KUKA KRL program: ab_a_lta_st01_g08.src, ab_a_lta_st01_g08.dat

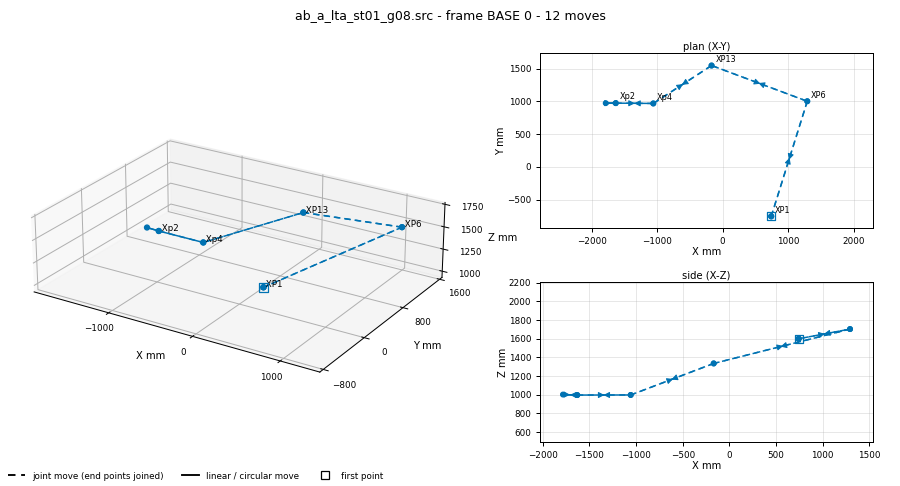
[picture p0: tool path of ab_a_lta_st01_g08.src in frame BASE 0, 12 of 12 moves have a stored position in this frame; points joined in program order, loops and branches not executed]
--- ab_a_lta_st01_g08.src ---
&ACCESS RVP1
&REL 10
&PARAM DISKPATH = KRC:\R1\Program\AXOR_ATEGO
DEF ab_a_lta_st01_g08( )

;FOLD INI;%{PE}
  ;FOLD BASISTECH INI
    GLOBAL INTERRUPT DECL 3 WHEN $STOPMESS==TRUE DO IR_STOPM ( )
    INTERRUPT ON 3
    BAS (#INITMOV,0 )
  ;ENDFOLD (BASISTECH INI)
;FOLD SPOTTECH INI
USERSPOT(#INIT)
;ENDFOLD (SPOTTECH INI)
;FOLD GRIPPERTECH INI
USER_GRP(0,DUMMY,DUMMY,GDEFAULT)
;ENDFOLD (GRIPPERTECH INI)
  ;FOLD USER INI
    ;Make your modifications here

  ;ENDFOLD (USER INI)
;ENDFOLD (INI)

;FOLD PTP P1 Vel=100 % PDAT1 Tool[5]:Gripper Geo G01 00 Base[0];%{PE}%R 8.2.24,%MKUKATPBASIS,%CMOVE,%VPTP,%P 1:PTP, 2:P1, 3:, 5:100, 7:PDAT1
$BWDSTART=FALSE
PDAT_ACT=PPDAT1
FDAT_ACT=FP1
BAS(#PTP_PARAMS,100)
PTP XP1
;ENDFOLD

; Caracterizacao dos meios de producao
; Changes: Deposita na Geo - ATEGO LTA
; Versao Atual: 28/12/2016
; Ferramenta: GRIPPER ATEGO/AXOR
; Name: P13.090-R6

chk_w5_wechs_ok ( )  ; CHECK GRP ATEGO

;FOLD PTP P5 Vel=100 % PDAT3 Tool[5]:Gripper Geo G01 00 Base[0];%{PE}%R 8.2.24,%MKUKATPBASIS,%CMOVE,%VPTP,%P 1:PTP, 2:P5, 3:, 5:100, 7:PDAT3
$BWDSTART=FALSE
PDAT_ACT=PPDAT3
FDAT_ACT=FP5
BAS(#PTP_PARAMS,100)
PTP XP5
;ENDFOLD

;FOLD ; Check Gripper GRAMPOS ABERTOS;%{PE}%R 8.2.24,%MKUKATPBASIS,%CCOMMENT,%VNORMAL,%P 2:Check Gripper GRAMPOS ABERTOS
;ENDFOLD
chk_w5_grp1_opn ()
chk_w5_grp2_opn ()
chk_w5_grp3_opn ()
chk_w5_grp4_opn ()

;FOLD ; Verifica GRIPPER SEM PECA;%{PE}%R 8.2.24,%MKUKATPBASIS,%CCOMMENT,%VNORMAL,%P 2:Verifica GRIPPER SEM PECA
;ENDFOLD
;FOLD WAIT FOR ( NOT IN 497 'Presenca peca 1 Axor/Atego' );%{PE}%R 8.2.24,%MKUKATPBASIS,%CEXT_WAIT_FOR,%VEXT_WAIT_FOR,%P 2:, 4:NOT, 5:$IN, 6:497, 7:Presenca peca 1 Axor/Atego, 9:
WAIT FOR  (  NOT $IN[497] )
;ENDFOLD
;FOLD WAIT FOR ( NOT IN 498 'Presenca peca 2 Axor/Atego' );%{PE}%R 8.2.24,%MKUKATPBASIS,%CEXT_WAIT_FOR,%VEXT_WAIT_FOR,%P 2:, 4:NOT, 5:$IN, 6:498, 7:Presenca peca 2 Axor/Atego, 9:
WAIT FOR  (  NOT $IN[498] )
;ENDFOLD

;FOLD ; Aguarda Liberacao p/ Encaixar no Painel Frontal ou Adiantamento;%{PE}%R 8.2.24,%MKUKATPBASIS,%CCOMMENT,%VNORMAL,%P 2:Aguarda Liberacao p/ Encaixar no  Painel Frontal ou Adiantamento
;ENDFOLD
;FOLD OUT 3347 'MAGAZINE 1 OCUPADO' State=TRUE ;%{PE}%R 8.2.24,%MKUKATPBASIS,%COUT,%VOUTX,%P 2:3347, 3:MAGAZINE 1 OCUPADO, 5:TRUE, 6:
$OUT[3347]=TRUE
;ENDFOLD
;FOLD OUT 3344 'APLICAÇÃO NÃO OK' State=TRUE ;%{PE}%R 8.2.24,%MKUKATPBASIS,%COUT,%VOUTX,%P 2:3344, 3:APLICAÇÃO NÃO OK, 5:TRUE, 6:
$OUT[3344]=TRUE
;ENDFOLD
;FOLD WAIT FOR ( IN 3347 'LIB. ANTECIPACAO (ATEGO/AXOR)' );%{PE}%R 8.2.24,%MKUKATPBASIS,%CEXT_WAIT_FOR,%VEXT_WAIT_FOR,%P 2:, 4:, 5:$IN, 6:3347, 7:LIB. ANTECIPACAO (ATEGO/AXOR), 9:
WAIT FOR  ( $IN[3347] )
;ENDFOLD
;FOLD OUT 3347 'MAGAZINE 1 OCUPADO' State=FALSE ;%{PE}%R 8.2.24,%MKUKATPBASIS,%COUT,%VOUTX,%P 2:3347, 3:MAGAZINE 1 OCUPADO, 5:FALSE, 6:
$OUT[3347]=FALSE
;ENDFOLD

;FOLD PTP P6 CONT Vel=100 % PDAT4 Tool[5]:Gripper Geo G01 00 Base[0];%{PE}%R 8.2.24,%MKUKATPBASIS,%CMOVE,%VPTP,%P 1:PTP, 2:P6, 3:C_PTP, 5:100, 7:PDAT4
$BWDSTART=FALSE
PDAT_ACT=PPDAT4
FDAT_ACT=FP6
BAS(#PTP_PARAMS,100)
PTP XP6 C_PTP
;ENDFOLD
;FOLD PTP P13 CONT Vel=100 % PDAT5 Tool[5]:Gripper Geo G01 00 Base[0];%{PE}%R 8.2.24,%MKUKATPBASIS,%CMOVE,%VPTP,%P 1:PTP, 2:P13, 3:C_PTP, 5:100, 7:PDAT5
$BWDSTART=FALSE
PDAT_ACT=PPDAT5
FDAT_ACT=FP13
BAS(#PTP_PARAMS,100)
PTP XP13 C_PTP
;ENDFOLD
;FOLD PTP p4 CONT Vel=100 % P_OLP3 Tool[5]:Gripper Geo G01 00 Base[0];%{PE}%R 8.2.24,%MKUKATPBASIS,%CMOVE,%VPTP,%P 1:PTP, 2:p4, 3:C_PTP, 5:100, 7:P_OLP3
$BWDSTART=FALSE
PDAT_ACT=PP_OLP3
FDAT_ACT=Fp4
BAS(#PTP_PARAMS,100)
PTP Xp4 C_PTP
;ENDFOLD

;FOLD ; Aguarda Liberacao p/ Encaixar GRIPPER no Painel Frontal;%{PE}%R 8.2.24,%MKUKATPBASIS,%CCOMMENT,%VNORMAL,%P 2:Aguarda Liberacao p/ Encaixar GRIPPER no Painel Frontal
;ENDFOLD
;FOLD WAIT FOR ( IN 3344 'LIB.P/APOIO DO TETO (ATEGO/AXOR)' );%{PE}%R 8.2.24,%MKUKATPBASIS,%CEXT_WAIT_FOR,%VEXT_WAIT_FOR,%P 2:, 4:, 5:$IN, 6:3344, 7:LIB.P/APOIO DO TETO (ATEGO/AXOR), 9:
WAIT FOR  ( $IN[3344] )
;ENDFOLD
;FOLD OUT 3344 'APLICAÇÃO NÃO OK' State=FALSE ;%{PE}%R 8.2.24,%MKUKATPBASIS,%COUT,%VOUTX,%P 2:3344, 3:APLICAÇÃO NÃO OK, 5:FALSE, 6:
$OUT[3344]=FALSE
;ENDFOLD

;FOLD LIN p2 Vel=0.25 m/s L_OLP1 Tool[5]:Gripper Geo G01 00 Base[0];%{PE}%R 8.2.24,%MKUKATPBASIS,%CMOVE,%VLIN,%P 1:LIN, 2:p2, 3:, 5:0.25, 7:L_OLP1
$BWDSTART=FALSE
LDAT_ACT=LL_OLP1
FDAT_ACT=Fp2
BAS(#CP_PARAMS,0.25)
LIN Xp2
;ENDFOLD

;FOLD ; Posicao Geometria Gripper ATEGO/AXOR;%{PE}%R 8.2.24,%MKUKATPBASIS,%CCOMMENT,%VNORMAL,%P 2:Posicao Geometria Gripper ATEGO/AXOR
;ENDFOLD
;FOLD LIN P14 Vel=0.15 m/s CPDAT1 Tool[5]:Gripper Geo G01 00 Base[0];%{PE}%R 8.2.24,%MKUKATPBASIS,%CMOVE,%VLIN,%P 1:LIN, 2:P14, 3:, 5:0.15, 7:CPDAT1
$BWDSTART=FALSE
LDAT_ACT=LCPDAT1
FDAT_ACT=FP14
BAS(#CP_PARAMS,0.15)
LIN XP14
;ENDFOLD

;FOLD ; Fechar Grampos Z4,Z2 e Z1;%{PE}%R 8.2.24,%MKUKATPBASIS,%CCOMMENT,%VNORMAL,%P 2:Fechar Grampos Z4,Z2 e Z1
;ENDFOLD
;FOLD SET GRP 4 State=CLO GDAT6;%{PE}%R 8.2.4,%MKUKATPGRP,%CGRP,%VGRP,%P 2:4, 4:1, 5:#NO, 6:GDAT6, 8:0, 10:0
H50(GRP,4,1,GGDAT6)
;ENDFOLD
chk_w5_grp4_clo ()
;FOLD SET GRP 1 State=CLO GDAT2;%{PE}%R 8.2.4,%MKUKATPGRP,%CGRP,%VGRP,%P 2:1, 4:1, 5:#NO, 6:GDAT2, 8:0, 10:0
H50(GRP,1,1,GGDAT2)
;ENDFOLD
;FOLD SET GRP 2 State=CLO GDAT3;%{PE}%R 8.2.4,%MKUKATPGRP,%CGRP,%VGRP,%P 2:2, 4:1, 5:#NO, 6:GDAT3, 8:0, 10:0
H50(GRP,2,1,GGDAT3)
;ENDFOLD
;FOLD ; Aguarda Grampos Z1 e Z2 FECHADOS e Z3 ABERTO;%{PE}%R 8.2.24,%MKUKATPBASIS,%CCOMMENT,%VNORMAL,%P 2:Aguarda Grampos Z1 e Z2 FECHADOS e Z3 ABERTO
;ENDFOLD
chk_w5_grp1_clo ()
chk_w5_grp2_clo ()
chk_w5_grp3_opn ()

;FOLD ; Verifica garra com peca;%{PE}%R 8.2.24,%MKUKATPBASIS,%CCOMMENT,%VNORMAL,%P 2:Verifica  garra  com  peca
;ENDFOLD
IF (NOT(GHOST())) THEN
;FOLD WAIT FOR ( IN 497 'Presenca peca 1 Axor/Atego' );%{PE}%R 8.2.24,%MKUKATPBASIS,%CEXT_WAIT_FOR,%VEXT_WAIT_FOR,%P 2:, 4:, 5:$IN, 6:497, 7:Presenca peca 1 Axor/Atego, 9:
WAIT FOR  ( $IN[497] )
;ENDFOLD
;FOLD WAIT FOR ( IN 498 'Presenca peca 2 Axor/Atego' );%{PE}%R 8.2.24,%MKUKATPBASIS,%CEXT_WAIT_FOR,%VEXT_WAIT_FOR,%P 2:, 4:, 5:$IN, 6:498, 7:Presenca peca 2 Axor/Atego, 9:
WAIT FOR  ( $IN[498] )
;ENDFOLD
ENDIF

;FOLD ; Robo na posicao;%{PE}%R 8.2.24,%MKUKATPBASIS,%CCOMMENT,%VNORMAL,%P 2:Robo  na  posicao
;ENDFOLD
;FOLD OUT 3345 'ALERTA DE APLICAÇÃO' State=TRUE ;%{PE}%R 8.2.24,%MKUKATPBASIS,%COUT,%VOUTX,%P 2:3345, 3:ALERTA DE APLICAÇÃO, 5:TRUE, 6:
$OUT[3345]=TRUE
;ENDFOLD

;FOLD ; Aguarda liberacao para sair com a garra;%{PE}%R 8.2.24,%MKUKATPBASIS,%CCOMMENT,%VNORMAL,%P 2:Aguarda  liberacao  para  sair  com  a  garra
;ENDFOLD
;FOLD WAIT FOR ( IN 3345 'LIB.SAÍDA APOIO DO TETO (ATEGO/AXOR)' );%{PE}%R 8.2.24,%MKUKATPBASIS,%CEXT_WAIT_FOR,%VEXT_WAIT_FOR,%P 2:, 4:, 5:$IN, 6:3345, 7:LIB.SAÍDA APOIO DO TETO (ATEGO/AXOR), 9:
WAIT FOR  ( $IN[3345] )
;ENDFOLD
;FOLD OUT 3345 'ALERTA DE APLICAÇÃO' State=FALSE ;%{PE}%R 8.2.24,%MKUKATPBASIS,%COUT,%VOUTX,%P 2:3345, 3:ALERTA DE APLICAÇÃO, 5:FALSE, 6:
$OUT[3345]=FALSE
;ENDFOLD

;FOLD ; Abrir grampos Z1,Z2,Z4;%{PE}%R 8.2.24,%MKUKATPBASIS,%CCOMMENT,%VNORMAL,%P 2:Abrir  grampos  Z1,Z2,Z4
;ENDFOLD
;FOLD SET GRP 1 State=OPN GDAT1;%{PE}%R 8.2.4,%MKUKATPGRP,%CGRP,%VGRP,%P 2:1, 4:2, 5:#NO, 6:GDAT1, 8:0, 10:0
H50(GRP,1,2,GGDAT1)
;ENDFOLD
;FOLD SET GRP 2 State=OPN GDAT7;%{PE}%R 8.2.4,%MKUKATPGRP,%CGRP,%VGRP,%P 2:2, 4:2, 5:#NO, 6:GDAT7, 8:0, 10:0
H50(GRP,2,2,GGDAT7)
;ENDFOLD
;FOLD SET GRP 3 State=OPN GDAT8;%{PE}%R 8.2.4,%MKUKATPGRP,%CGRP,%VGRP,%P 2:3, 4:2, 5:#NO, 6:GDAT8, 8:0, 10:0
H50(GRP,3,2,GGDAT8)
;ENDFOLD
;FOLD SET GRP 4 State=OPN GDAT9;%{PE}%R 8.2.4,%MKUKATPGRP,%CGRP,%VGRP,%P 2:4, 4:2, 5:#NO, 6:GDAT9, 8:0, 10:0
H50(GRP,4,2,GGDAT9)
;ENDFOLD
chk_w5_grp1_opn ()
chk_w5_grp2_opn ()
chk_w5_grp3_opn ()
chk_w5_grp4_opn ()

;FOLD LIN P15 Vel=0.15 m/s CPDAT2 Tool[5]:Gripper Geo G01 00 Base[0];%{PE}%R 8.2.24,%MKUKATPBASIS,%CMOVE,%VLIN,%P 1:LIN, 2:P15, 3:, 5:0.15, 7:CPDAT2
$BWDSTART=FALSE
LDAT_ACT=LCPDAT2
FDAT_ACT=FP15
BAS(#CP_PARAMS,0.15)
LIN XP15
;ENDFOLD

;FOLD WAIT FOR ( NOT IN 497 'Presenca peca 1 Axor/Atego' );%{PE}%R 8.2.24,%MKUKATPBASIS,%CEXT_WAIT_FOR,%VEXT_WAIT_FOR,%P 2:, 4:NOT, 5:$IN, 6:497, 7:Presenca peca 1 Axor/Atego, 9:
WAIT FOR  (  NOT $IN[497] )
;ENDFOLD
;FOLD WAIT FOR ( NOT IN 498 'Presenca peca 2 Axor/Atego' );%{PE}%R 8.2.24,%MKUKATPBASIS,%CEXT_WAIT_FOR,%VEXT_WAIT_FOR,%P 2:, 4:NOT, 5:$IN, 6:498, 7:Presenca peca 2 Axor/Atego, 9:
WAIT FOR  (  NOT $IN[498] )
;ENDFOLD

;FOLD PTP P0 Vel=100 % P_OLP7 Tool[5]:Gripper Geo G01 00 Base[0];%{PE}%R 8.2.24,%MKUKATPBASIS,%CMOVE,%VPTP,%P 1:PTP, 2:P0, 3:, 5:100, 7:P_OLP7
$BWDSTART=FALSE
PDAT_ACT=PP_OLP7
FDAT_ACT=FP0
BAS(#PTP_PARAMS,100)
PTP XP0
;ENDFOLD
;FOLD PTP p9 CONT Vel=100 % P_OLP5 Tool[5]:Gripper Geo G01 00 Base[0];%{PE}%R 8.2.24,%MKUKATPBASIS,%CMOVE,%VPTP,%P 1:PTP, 2:p9, 3:C_PTP, 5:100, 7:P_OLP5
$BWDSTART=FALSE
PDAT_ACT=PP_OLP5
FDAT_ACT=Fp9
BAS(#PTP_PARAMS,100)
PTP Xp9 C_PTP
;ENDFOLD
;FOLD PTP p12 CONT Vel=100 % P_OLP6 Tool[5]:Gripper Geo G01 00 Base[0];%{PE}%R 8.2.24,%MKUKATPBASIS,%CMOVE,%VPTP,%P 1:PTP, 2:p12, 3:C_PTP, 5:100, 7:P_OLP6
$BWDSTART=FALSE
PDAT_ACT=PP_OLP6
FDAT_ACT=Fp12
BAS(#PTP_PARAMS,100)
PTP Xp12 C_PTP
;ENDFOLD
;FOLD PTP P16 Vel=100 % PDAT6 Tool[5]:Gripper Geo G01 00 Base[0];%{PE}%R 8.2.24,%MKUKATPBASIS,%CMOVE,%VPTP,%P 1:PTP, 2:P16, 3:, 5:100, 7:PDAT6
$BWDSTART=FALSE
PDAT_ACT=PPDAT6
FDAT_ACT=FP16
BAS(#PTP_PARAMS,100)
PTP XP16
;ENDFOLD

;FOLD ; Libera dispositivo para soldar respot;%{PE}%R 8.2.24,%MKUKATPBASIS,%CCOMMENT,%VNORMAL,%P 2:Libera  dispositivo  para  soldar  respot
;ENDFOLD
;FOLD OUT 3347 'MAGAZINE 1 OCUPADO' State=TRUE ;%{PE}%R 8.2.24,%MKUKATPBASIS,%COUT,%VOUTX,%P 2:3347, 3:MAGAZINE 1 OCUPADO, 5:TRUE, 6:
$OUT[3347]=TRUE
;ENDFOLD
;FOLD OUT 3344 'APLICAÇÃO NÃO OK' State=TRUE ;%{PE}%R 8.2.24,%MKUKATPBASIS,%COUT,%VOUTX,%P 2:3344, 3:APLICAÇÃO NÃO OK, 5:TRUE, 6:
$OUT[3344]=TRUE
;ENDFOLD

;FOLD PULSE 3340 'R6 GEOMETRIA OK' State=TRUE Time=1 sec;%{PE}%R 8.2.24,%MKUKATPBASIS,%COUT,%VPULSE,%P 2:3340, 3:R6 GEOMETRIA OK, 5:TRUE, 6:, 8:1
PULSE($OUT[3340], TRUE,1)
;ENDFOLD
END

--- ab_a_lta_st01_g08.dat ---
&ACCESS RVP1
&REL 10
&PARAM DISKPATH = KRC:\R1\Program\AXOR_ATEGO
DEFDAT  ab_a_lta_st01_g08
;FOLD EXTERNAL DECLARATIONS;%{PE}%MKUKATPBASIS,%CEXT,%VCOMMON,%P
;FOLD BASISTECH EXT;%{PE}%MKUKATPBASIS,%CEXT,%VEXT,%P
EXT  BAS (BAS_COMMAND  :IN,REAL  :IN )
DECL INT SUCCESS
;ENDFOLD (BASISTECH EXT)
;FOLD USER EXT;%{E}%MKUKATPUSER,%CEXT,%VEXT,%P
;Make your modifications here
;ENDFOLD (USER EXT)
;ENDFOLD (EXTERNAL DECLARATIONS)

;# ============ START PATH : ab_a_lta_st01_g08 =============
DECL FDAT Fp11={TOOL_NO 5,BASE_NO 0,IPO_FRAME #BASE,POINT2[] " "}
DECL PDAT PP_OLP1={VEL 100.0,ACC 100.0,APO_DIST 0.0}
DECL E6POS Xp11={X 1293.05103,Y 1000.521,Z 1703.34399,A 36.1688995,B -6.9552002,C 153.792801,S 6,T 19}
DECL FDAT Fp10={TOOL_NO 5,BASE_NO 0,IPO_FRAME #BASE,POINT2[] " "}
DECL PDAT PP_OLP2={VEL 100.0,ACC 100.0,APO_DIST 0.0}
DECL E6POS Xp10={X -168.237,Y 1546.06995,Z 1335.04004,A 110.0187,B -0.406599998,C 159.128998,S 6,T 19}
DECL FDAT Fp4={TOOL_NO 5,BASE_NO 0,IPO_FRAME #BASE,POINT2[] " "}
DECL PDAT PP_OLP3={VEL 100.0,ACC 20.0,APO_DIST 0.0,APO_MODE #CPTP}
DECL E6POS Xp4={X -1057.83704,Y 966.953003,Z 997.169983,A -179.672195,B -1.48539996,C 179.896301,S 6,T 19}
DECL FDAT Fp2={TOOL_NO 5,BASE_NO 0,IPO_FRAME #BASE,POINT2[] " "}
DECL E6POS Xp2={X -1631.20996,Y 971.839417,Z 996.094482,A -179.828995,B -0.654202104,C 179.611496,S 22,T 19,E1 0.0,E2 0.0,E3 0.0,E4 0.0,E5 0.0,E6 0.0}
DECL LDAT LL_OLP1={VEL 0.25,ACC 100.0,APO_DIST 0.0,APO_FAC 0.0,ORI_TYP #VAR,CIRC_TYP #BASE,JERK_FAC 50.0}
DECL FDAT Fl005={TOOL_NO 5,BASE_NO 0,IPO_FRAME #BASE,POINT2[] " "}
DECL E6POS Xl005={X -1795.66003,Y 969.495972,Z 1016.79303,A 179.821594,B -1.35329998,C 179.764893,S 6,T 19}
DECL LDAT LL_OLP2={VEL 0.100000001,ACC 100.0,APO_DIST 0.0,APO_FAC 0.0,ORI_TYP #VAR,CIRC_TYP #BASE,JERK_FAC 50.0}
DECL FDAT Fp7={TOOL_NO 5,BASE_NO 0,IPO_FRAME #BASE,POINT2[] " "}
DECL E6POS Xp7={X -1650.26294,Y 963.580017,Z 1010.07397,A -179.672302,B -1.48520005,C 179.896301,S 6,T 19}
DECL LDAT LL_OLP3={VEL 0.25,ACC 100.0,APO_DIST 0.0,APO_FAC 0.0,ORI_TYP #VAR,CIRC_TYP #BASE,JERK_FAC 50.0}
DECL FDAT Fp8={TOOL_NO 5,BASE_NO 0,IPO_FRAME #BASE,POINT2[] " "}
DECL PDAT PP_OLP4={VEL 100.0,ACC 100.0,APO_DIST 0.0}
DECL E6POS Xp8={X -1057.83704,Y 966.953003,Z 997.169983,A -179.672302,B -1.48539996,C 179.896301,S 6,T 19}
DECL FDAT Fp9={TOOL_NO 5,BASE_NO 0,IPO_FRAME #BASE,POINT2[] " "}
DECL PDAT PP_OLP5={VEL 100.0,ACC 20.0,APO_DIST 20.0,APO_MODE #CPTP}
DECL E6POS Xp9={X -168.237,Y 1546.06995,Z 1335.04004,A 110.0187,B -0.406599998,C 159.128998,S 6,T 19}
DECL FDAT Fp12={TOOL_NO 5,BASE_NO 0,IPO_FRAME #BASE,POINT2[] " "}
DECL PDAT PP_OLP6={VEL 100.0,ACC 20.0,APO_DIST 20.0,APO_MODE #CPTP}
DECL E6POS Xp12={X 1293.05103,Y 1000.521,Z 1703.34399,A 36.1688995,B -6.9552002,C 153.792801,S 6,T 19}
DECL BASIS_SUGG_T LAST_BASIS={POINT1[] "P0                      ",POINT2[] "P0                      ",CP_PARAMS[] "CPDAT0                  ",PTP_PARAMS[] "PDAT0                   ",CONT[] "                        ",CP_VEL[] "2.0                     ",PTP_VEL[] "100                     ",SYNC_PARAMS[] "SYNCDAT                 ",SPL_NAME[] "S0                      "}
DECL E6POS XP1={X 743.006714,Y -756.668091,Z 1599.74805,A -36.0596199,B 42.8596992,C 82.0244064,S 18,T 2,E1 0.0,E2 0.0,E3 0.0,E4 0.0,E5 0.0,E6 0.0}
DECL FDAT FP1={TOOL_NO 5,BASE_NO 0,IPO_FRAME #BASE,POINT2[] " ",TQ_STATE FALSE}
DECL PDAT PPDAT1={VEL 100.0,ACC 20.0,APO_DIST 100.0,GEAR_JERK 50.0}
DECL E6POS XP3={X 742.632385,Y -756.358521,Z 1599.651,A -36.0531197,B 42.8928986,C 82.0324936,S 18,T 2,E1 0.0,E2 0.0,E3 0.0,E4 0.0,E5 0.0,E6 0.0}
DECL FDAT FP3={TOOL_NO 5,BASE_NO 0,IPO_FRAME #BASE,POINT2[] " ",TQ_STATE FALSE}
DECL PDAT PPDAT2={VEL 100.0,ACC 100.0,APO_DIST 100.0,GEAR_JERK 50.0}
DECL E6POS XP5={X 742.628418,Y -756.355896,Z 1599.65405,A -36.0531693,B 42.8930511,C 82.0323792,S 18,T 2,E1 0.0,E2 0.0,E3 0.0,E4 0.0,E5 0.0,E6 0.0}
DECL FDAT FP5={TOOL_NO 5,BASE_NO 0,IPO_FRAME #BASE,POINT2[] " ",TQ_STATE FALSE}
DECL PDAT PPDAT3={VEL 100.0,ACC 20.0,APO_DIST 100.0,GEAR_JERK 50.0}
DECL E6POS XP6={X 1293.05103,Y 1000.526,Z 1703.34595,A 36.1689301,B -6.95535898,C 153.792694,S 22,T 19,E1 0.0,E2 0.0,E3 0.0,E4 0.0,E5 0.0,E6 0.0}
DECL FDAT FP6={TOOL_NO 5,BASE_NO 0,IPO_FRAME #BASE,POINT2[] " ",TQ_STATE FALSE}
DECL PDAT PPDAT4={VEL 100.0,ACC 20.0,APO_DIST 20.0,APO_MODE #CPTP,GEAR_JERK 50.0}
DECL E6POS XP13={X -168.237503,Y 1546.06799,Z 1335.04297,A 110.018799,B -0.406741798,C 159.129105,S 22,T 19,E1 0.0,E2 0.0,E3 0.0,E4 0.0,E5 0.0,E6 0.0}
DECL FDAT FP13={TOOL_NO 5,BASE_NO 0,IPO_FRAME #BASE,POINT2[] " ",TQ_STATE FALSE}
DECL PDAT PPDAT5={VEL 100.0,ACC 20.0,APO_DIST 20.0,APO_MODE #CPTP,GEAR_JERK 50.0}
DECL GRP_SUGG_T LAST_GRP={NUMBER[] "3                       ",STATE[] "1                       ",PARAMS[] "GDAT11                  "}
DECL GRP_TYP GGDAT1={G_APO #NO,GRP_TIME 0.200000003,CTRL #OFF,DLY 0,DST 1}
DECL GRP_TYP GGDAT2={G_APO #NO,GRP_TIME 0.200000003,CTRL #OFF,DLY 0,DST 1}
DECL GRP_TYP GGDAT3={G_APO #NO,GRP_TIME 0.200000003,CTRL #OFF,DLY 0,DST 1}
DECL GRP_TYP GCONT={G_APO #YES,GRP_TIME 0.0,CTRL #OFF,DLY 0,DST 0}
DECL GRP_TYP GGDAT4={G_APO #NO,GRP_TIME 0.200000003,CTRL #OFF,DLY 0,DST 1}
DECL E6POS XP14={X -1784.052,Y 971.415588,Z 1001.565,A -179.827499,B -0.651935518,C 179.6091,S 22,T 19,E1 0.0,E2 0.0,E3 0.0,E4 0.0,E5 0.0,E6 0.0}
DECL FDAT FP14={TOOL_NO 5,BASE_NO 0,IPO_FRAME #BASE,POINT2[] " ",TQ_STATE FALSE}
DECL LDAT LCPDAT1={VEL 2.0,ACC 100.0,APO_DIST 100.0,APO_FAC 50.0,AXIS_VEL 100.0,AXIS_ACC 100.0,ORI_TYP #VAR,CIRC_TYP #BASE,JERK_FAC 50.0,GEAR_JERK 50.0,EXAX_IGN 0}
DECL GRP_TYP GGDAT5={G_APO #NO,GRP_TIME 0.200000003,CTRL #OFF,DLY 0,DST 1}
DECL E6POS XP15={X -1631.19897,Y 971.837219,Z 996.094604,A -179.828796,B -0.654016376,C 179.611496,S 22,T 19,E1 0.0,E2 0.0,E3 0.0,E4 0.0,E5 0.0,E6 0.0}
DECL FDAT FP15={TOOL_NO 5,BASE_NO 0,IPO_FRAME #BASE,POINT2[] " ",TQ_STATE FALSE}
DECL LDAT LCPDAT2={VEL 2.0,ACC 100.0,APO_DIST 100.0,APO_FAC 50.0,AXIS_VEL 100.0,AXIS_ACC 100.0,ORI_TYP #VAR,CIRC_TYP #BASE,JERK_FAC 50.0,GEAR_JERK 50.0,EXAX_IGN 0}
DECL PDAT PP_OLP7={VEL 100.0,ACC 20.0,APO_DIST 0.0}
DECL E6POS XP0={X -1057.83704,Y 966.953003,Z 997.169983,A -179.672302,B -1.48539996,C 179.896301,S 6,T 19}
DECL FDAT FP0={TOOL_NO 5,BASE_NO 0,IPO_FRAME #BASE,POINT2[] " "}
DECL E6POS XP16={X 743.061279,Y -756.612671,Z 1599.71704,A -36.059021,B 42.8573494,C 82.0305023,S 18,T 2,E1 0.0,E2 0.0,E3 0.0,E4 0.0,E5 0.0,E6 0.0}
DECL FDAT FP16={TOOL_NO 5,BASE_NO 0,IPO_FRAME #BASE,POINT2[] " ",TQ_STATE FALSE}
DECL PDAT PPDAT6={VEL 100.0,ACC 20.0,APO_DIST 100.0,APO_MODE #CPTP,GEAR_JERK 50.0}
DECL GRP_TYP GGDAT6={G_APO #NO,GRP_TIME 0.200000003,CTRL #OFF,DLY 0,DST 1}
DECL GRP_TYP GGDAT7={G_APO #NO,GRP_TIME 0.200000003,CTRL #OFF,DLY 0,DST 1}
DECL GRP_TYP GGDAT8={G_APO #NO,GRP_TIME 0.200000003,CTRL #OFF,DLY 0,DST 1}
DECL GRP_TYP GGDAT9={G_APO #NO,GRP_TIME 0.200000003,CTRL #OFF,DLY 0,DST 1}
DECL GRP_TYP GGDAT10={G_APO #NO,GRP_TIME 0.200000003,CTRL #OFF,DLY 0,DST 1}
DECL GRP_TYP GGDAT11={G_APO #NO,GRP_TIME 0.200000003,CTRL #OFF,DLY 0,DST 1}
ENDDAT
